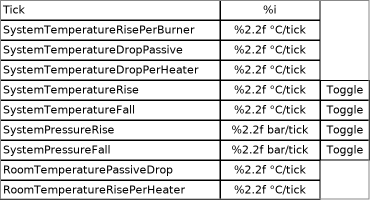
VISUALIZATION UI_Sim  // 370x200
VAR_IN_OUT
	param			: SimulationGlobalParameters;
END_VAR
    Rectangle (220,40 100x20), "%2.2f °C/tick", text variable: param.rSystemTemperatureDropPassive
        OnMouseClick: write the text variable via Default
    Rectangle (0,20 220x20), "SystemTemperatureRisePerBurner"
    Rectangle (220,20 100x20), "%2.2f °C/tick", text variable: param.rSystemTemperatureRisePerBurner
        OnMouseClick: write the text variable via Default
    Rectangle (0,40 220x20), "SystemTemperatureDropPassive"
    Rectangle (0,60 220x20), "SystemTemperatureDropPerHeater"
    Rectangle (0,80 220x20), "SystemTemperatureRise"
    Rectangle (0,100 220x20), "SystemTemperatureFall"
    Rectangle (0,120 220x20), "SystemPressureRise"
    Rectangle (0,140 220x20), "SystemPressureFall"
    Rectangle (0,160 220x20), "RoomTemperaturePassiveDrop"
    Rectangle (0,180 220x20), "RoomTemperatureRisePerHeater"
    Rectangle (220,80 100x20), "%2.2f °C/tick", text variable: param.rSystemTemperatureRise
        OnMouseClick: write the text variable via Default
    Rectangle (220,60 100x20), "%2.2f °C/tick", text variable: param.rSystemTemperatureDropPerHeater
        OnMouseClick: write the text variable via Default
    Rectangle (220,120 100x20), "%2.2f bar/tick", text variable: param.rSystemPressureRise
        OnMouseClick: write the text variable via Default
    Rectangle (220,100 100x20), "%2.2f °C/tick", text variable: param.rSystemTemperatureFall
        OnMouseClick: write the text variable via Default
    Rectangle (220,160 100x20), "%2.2f °C/tick", text variable: param.rRoomTemperaturePassiveDrop
        OnMouseClick: write the text variable via Default
    Rectangle (220,140 100x20), "%2.2f bar/tick", text variable: param.rSystemPressureFall
        OnMouseClick: write the text variable via Default
    Rectangle (220,180 100x20), "%2.2f °C/tick", text variable: param.rRoomTemperatureRisePerHeater
        OnMouseClick: write the text variable via Default
    Rectangle (0,0 220x20), "Tick"
    Rectangle (220,0 100x20), "%i", text variable: param.nTick
        OnMouseClick: write the text variable via Default
    Rectangle (320,80 50x20), "Toggle", text variable: param.bToggleSystemTemperatureRise
        toggle param.bToggleSystemTemperatureRise
    Rectangle (320,100 50x20), "Toggle", text variable: param.bToggleSystemTemperatureFall
        toggle param.bToggleSystemTemperatureFall
    Rectangle (320,120 50x20), "Toggle", text variable: param.bToggleSystemPressureRise
        toggle param.bToggleSystemPressureRise
    Rectangle (320,140 50x20), "Toggle", text variable: param.bToggleSystemPressureFall
        toggle param.bToggleSystemPressureFall
END_VISUALIZATION

(* stored: Version 1.1.0.1
   Visu UI_Sim: Id {6c9dfb51-5ace-4849-a9a8-b6e8362802a6} *)
